// TwinCAT 3 PLC project PLC
// ProgramVersion: 3.1.4023.0
// libraries:
//   Tc2_ControllerToolbox, * (Beckhoff Automation GmbH)
//   Tc2_MC2, * (Beckhoff Automation GmbH)
//   Tc2_ModbusRTU, * (Beckhoff Automation GmbH)
//   Tc2_ModbusSrv, * (Beckhoff Automation GmbH)
//   Tc2_SerialCom, * (Beckhoff Automation GmbH)
//   Tc2_Standard, * (Beckhoff Automation GmbH)
//   Tc2_System, * (Beckhoff Automation GmbH)
//   Tc2_Utilities, * (Beckhoff Automation GmbH)
//   Tc3_Module, * (Beckhoff Automation GmbH)
//   VisuDialogs, * (System)
//   VisuSymbols,3.5.10.0,System
// project tree:
//   DUTs/ DUT_MB.TcDUT, DUT_MBReads.TcDUT
//   / Fast.TcTTO, GlobalTextList.TcGTLO, PlcTask.TcTTO, Visualization Manager.TcVMO (not stored)
//   GVLs/ GVL.TcGVL
//   POUs/ Background.TcPOU, BackgroundEL.TcPOU, FB_CCMT4Setup.TcPOU, FB_FanModbus.TcPOU, FB_FanWriteReg.TcPOU, FB_FormatTempRTD.TcPOU, FB_FormatTempTC.TcPOU, FB_LedOff.TcPOU, FB_ModBusTCPReadRegs.TcPOU, FB_ValveModbus.TcPOU, FB_MoveStepperRel.TcPOU, FB_MoveStepperLoop.TcPOU, FB_MoveStepperAbs.TcPOU, FB_mVtoTemp.TcPOU, FB_PLoop.TcPOU, FB_SanityCheck.TcPOU, FB_SerialCom.TcPOU, FB_StepperCtrl.TcPOU, FB_ModBusTCPWriteRegs.TcPOU, MAIN.TcPOU
//   VISUs/ Visu_MAIN.TcVIS

CONFIGURATION PLC
    RESOURCE PLC ON TwinCAT3
        TASK Fast(INTERVAL := T#1ms, PRIORITY := 4);
        TASK PlcTask(INTERVAL := T#10ms, PRIORITY := 10);
        PROGRAM Background WITH Fast : Background;
        PROGRAM MAIN WITH PlcTask : MAIN;
    END_RESOURCE
END_CONFIGURATION

// ---- DUTs/DUT_MB.TcDUT
TYPE DUT_MB :
STRUCT
	
	bExecute	:BOOL;	
	bBusy		:BOOL;
	bError		:BOOL;
	nErrId		:UDINT;
	
END_STRUCT
END_TYPE

// ---- DUTs/DUT_MBReads.TcDUT
TYPE DUT_MBReads EXTENDS DUT_MB :
STRUCT
	cbRead:UDINT;
	
END_STRUCT
END_TYPE

// ---- GVLs/GVL.TcGVL
VAR_GLOBAL
	RxBufferEL_RTD				: ComBuffer;		(* Receive data buffer; used with all receive function blocks *)
	TxBufferEL_RTD				: ComBuffer;		(* Transmit data buffer; used with all receive function blocks *)
	RxBufferEL_TC				: ComBuffer;		(* Receive data buffer; used with all receive function blocks *)
	TxBufferEL_TC				: ComBuffer;		(* Transmit data buffer; used with all receive function blocks *)
	RxBufferEL_Flow				: ComBuffer;
	TxBufferEL_Flow				: ComBuffer;
	RxBufferEL_MB				: ComBuffer;
	TxBufferEL_MB				: ComBuffer;
	f_mbMaster					: ModbusRtuMaster_KL6x22B;
	
	MAX_CSV_ROWS 				: UDINT := 100;
	MAX_CSV_COLUMNS 			: UDINT := 5;
	MAX_CSV_FIELD_LENGTH		: UDINT := 100;
(*	
// AXIS 1 CONTROL VARIABLES
	bEnable1				 	: BOOL := FALSE;	(* Axis enabled state *)
	bMove_Absolute1			 	: BOOL := FALSE;	(* Starts an absolute motion *)
	bJogFwd1				 	: BOOL := FALSE;	(* Starts rotating the axis at constant speed with CW direction *)
	bJogBack1				 	: BOOL := FALSE;	(* Starts rotating the axis at constant speed with CCCW direction *)
	bReset1					 	: BOOL := FALSE;	(* Resets the axis *)
	bHalt1					 	: BOOL := FALSE;	(* Stops the axis *)
	bStop1					 	: BOOL := FALSE;	(* Stops the axis *)
	bestop1					 	: BOOL := TRUE;		(* ESTOP button status *)
	bMove_Jog1				 	: BOOL := FALSE;	(* Starts actual motion *)
	bJogC1					 	: BOOL := FALSE;	(* Final Jog flag *)
	position1 					: UDINT;
	
// AXIS 2 CONTROL VARIABLES
	bEnable2				 	: BOOL := FALSE;	(* Axis enabled state *)
	bMove_Absolute2			 	: BOOL := FALSE;	(* Starts an absolute motion *)
	bJogFwd2				 	: BOOL := FALSE;	(* Starts rotating the axis at constant speed with CW direction *)
	bJogBack2				 	: BOOL := FALSE;	(* Starts rotating the axis at constant speed with CCCW direction *)
	bReset2					 	: BOOL := FALSE;	(* Resets the axis *)
	bHalt2					 	: BOOL := FALSE;	(* Stops the axis *)
	bStop2					 	: BOOL := FALSE;	(* Stops the axis *)
	bestop2					 	: BOOL := TRUE;		(* ESTOP button status *)
	bMove_Jog2				 	: BOOL := FALSE;	(* Starts actual motion *)
	bJogC2					 	: BOOL := FALSE;	(* Final Jog flag *)
	position2 					: UDINT;
*)	
// RELAY CONTROL VARIABLES
	bRelay1	AT %Q*			 	: BOOL := FALSE;
	bRelay2	AT %Q*				: BOOL := FALSE;
	
// 4...20mA ANALOG INPUT VARIABLES
	aiPress01 AT %I*			: INT;
	aiPress02 AT %I*			: INT;	
	aiPress03 AT %I*			: INT;	
	aiPress04 AT %I*			: INT;
	aiHBX01 AT %I*				: INT;
	
// RTD TEMPERATURE VARIABLES
	rtd01						: INT;
	rtd02						: INT;
	
// 0-10V ANALOG INPUT VARIABLES
	flow01 AT %I*				: INT;
	aiV02	AT %I*				: INT;
	
// PID VARIABLES
	TargetPos AT %Q*			: LREAL;
	
// 2Ch RTD VARIABLES
	RTD2Ch1	AT %I*				: INT;
	RTD2Ch2	AT %I*				: INT;
	RTD2Ch3	AT %I*				: INT;
	RTD2Ch4	AT %I*				: INT;
	RTD2Ch5	AT %I*				: INT;
	RTD2Ch6	AT %I*				: INT;
	RTD2Ch7	AT %I*				: INT;
	RTD2Ch8	AT %I*				: INT;
	
// 4Ch RTD VARIABLES
	RTD4Ch1	AT %I*				: INT;
	
END_VAR

// ---- POUs/Background.TcPOU
PROGRAM Background
VAR
END_VAR

(*
The SerialLineControl function block is supposed to be called in every PLC cycle.
It communicates with the serial line hardware device and transmits or receives data.
The SerialLineControl can be called in the standard task (e.g.for PcCOM port usage) 
or in a separate fast task (e.g.for terminal usage) as well.
A fast separate task will be necessary at high baud rates or with KL6001 terminals 
which have a small process image (3 or 5 data bytes only)
*)

(* background communication with the EL6002 and EL6021 terminal *)
BackgroundEL();

END_PROGRAM

// ---- POUs/BackgroundEL.TcPOU
PROGRAM BackgroundEL
VAR
	(* background communication with the EL6021 terminal *)
	fbEL6021Ctrl_RTD			: SerialLineControl;
	bEL6021CtrlError_RTD		: BOOL;
	eEL6021CtrlErrorID_RTD		: ComError_t;
	(* 	I/O variables for a EL6021 terminal*)
	stIn_EL6001_RTD AT %I*		: EL6inData22B;	(* linked to the EL6001 in the TwinCAT System Manager *)
	stOut_EL6001_RTD AT %Q*		: EL6outData22B;(* linked to the EL6001 in the TwinCAT System Manager *)
	
	(* background communication with the EL6021 terminal *)
	fbEL6021Ctrl_TC			: SerialLineControl;
	bEL6021CtrlError_TC		: BOOL;
	eEL6021CtrlErrorID_TC		: ComError_t;
	(* 	I/O variables for a EL6021 terminal*)
	stIn_EL6001_TC AT %I*		: EL6inData22B;	(* linked to the EL6001 in the TwinCAT System Manager *)
	stOut_EL6001_TC AT %Q*		: EL6outData22B;(* linked to the EL6001 in the TwinCAT System Manager *)
	
	(* background communication with the EL6002 terminal *)
	fbEL6002Ctrl_Flow			: SerialLineControl;
	bEL6002CtrlError_Flow		: BOOL;
	eEL6002CtrlErrorID_Flow		: ComError_t;
	(* 	I/O variables for a EL6002 terminal*)
	stIn_EL6002_Flow AT %I*		: EL6inData22B;	(* linked to the EL6001 in the TwinCAT System Manager *)
	stOut_EL6002_Flow AT %Q*		: EL6outData22B;(* linked to the EL6001 in the TwinCAT System Manager *)
	
		(* background communication with the EL6002 terminal *)
	fbEL6002Ctrl_MB			: SerialLineControl;
	bEL6002CtrlError_MB		: BOOL;
	eEL6002CtrlErrorID_MB		: ComError_t;
	(* 	I/O variables for a EL6002 terminal*)
	stIn_EL6002_MB AT %I*		: EL6inData22B;	(* linked to the EL6001 in the TwinCAT System Manager *)

END_VAR
VAR_INPUT
		stOut_EL6002_MB AT %Q*		: EL6outData22B;(* linked to the EL6001 in the TwinCAT System Manager *)
END_VAR

(*
The SerialLineControl function block is supposed to be called in every PLC cycle.
It communicates with the serial line hardware device and transmits or receives data.
The SerialLineControl can be called in the standard task (e.g.for PcCOM port usage) 
or in a separate fast task (e.g.for terminal usage) as well.
A fast separate task will be necessary at high baud rates or with KL6001 terminals 
which have a small process image (3 or 5 data bytes only)
*)

(* background communication with the EL6021 terminal *)
fbEL6021Ctrl_RTD(
	Mode := SERIALLINEMODE_EL6_22B,
	pComIn := ADR(stIn_EL6001_RTD), 
	pComOut:= ADR(stOut_EL6001_RTD), 
	SizeComIn := SIZEOF(stIn_EL6001_RTD), 
	Error => bEL6021CtrlError_RTD, 
	ErrorID => eEL6021CtrlErrorID_RTD,
	TxBuffer := GVL.TxBufferEL_RTD, 
	RxBuffer := GVL.RxBufferEL_RTD );
IF fbEL6021Ctrl_RTD.Error THEN
	bEL6021CtrlError_RTD := TRUE;
	eEL6021CtrlErrorID_RTD := fbEL6021Ctrl_RTD.ErrorID;
END_IF

(* background communication with the EL6021 terminal *)
fbEL6021Ctrl_TC(
	Mode := SERIALLINEMODE_EL6_22B,
	pComIn := ADR(stIn_EL6001_TC), 
	pComOut:= ADR(stOut_EL6001_TC), 
	SizeComIn := SIZEOF(stIn_EL6001_TC), 
	Error => bEL6021CtrlError_TC, 
	ErrorID => eEL6021CtrlErrorID_TC,
	TxBuffer := GVL.TxBufferEL_TC, 
	RxBuffer := GVL.RxBufferEL_TC );
IF fbEL6021Ctrl_TC.Error THEN
	bEL6021CtrlError_TC := TRUE;
	eEL6021CtrlErrorID_TC := fbEL6021Ctrl_RTD.ErrorID;
END_IF

(* background communication with the EL6021 terminal *)
fbEL6002Ctrl_Flow(
	Mode := SERIALLINEMODE_EL6_22B,
	pComIn := ADR(stIn_EL6002_Flow), 
	pComOut:= ADR(stOut_EL6002_Flow), 
	SizeComIn := SIZEOF(stIn_EL6002_Flow), 
	Error => bEL6002CtrlError_Flow, 
	ErrorID => eEL6002CtrlErrorID_Flow,
	TxBuffer := GVL.TxBufferEL_Flow, 
	RxBuffer := GVL.RxBufferEL_Flow );
IF fbEL6002Ctrl_Flow.Error THEN
	bEL6002CtrlError_Flow := TRUE;
	eEL6002CtrlErrorID_Flow := fbEL6002Ctrl_Flow.ErrorID;
END_IF

(* background communication with the EL6021 terminal *)
fbEL6002Ctrl_MB(
	Mode := SERIALLINEMODE_EL6_22B,
	pComIn := ADR(stIn_EL6002_MB), 
	pComOut:= ADR(stOut_EL6002_MB), 
	SizeComIn := SIZEOF(stIn_EL6002_MB), 
	Error => bEL6002CtrlError_MB, 
	ErrorID => eEL6002CtrlErrorID_MB,
	TxBuffer := GVL.TxBufferEL_MB, 
	RxBuffer := GVL.RxBufferEL_MB );
IF fbEL6002Ctrl_MB.Error THEN
	bEL6002CtrlError_MB := TRUE;
	eEL6002CtrlErrorID_MB := fbEL6002Ctrl_MB.ErrorID;
END_IF

END_PROGRAM

// ---- POUs/MAIN.TcPOU
PROGRAM MAIN
VAR
	fbEL6021RTD				: FB_SerialCom;
	fbEL6021TC				: FB_SerialCom;
	fbEL6002Flow			: FB_SerialCom;
	fbEL6021_MB				: FB_SerialCom;
	fbDoesItWork			: FB_SanityCheck;
	fbFormatRTD				: FB_FormatTempRTD;
	fbFormatTC				: FB_FormatTempTC;
	fbmVtoTemp				: FB_mVtoTemp;
	fbLedOff				: FB_LedOff;
	error					: ComError_t;
	fbPID					: FB_Ploop;
//	fbCloseValve1			: FB_CloseValve;
	fbMoveAxis1Rel			: FB_MoveStepperRel;
	fbMoveAxis1Abs			: FB_MoveStepperAbs;
	fbStepperLoop			: FB_MoveStepperLoop;
	
// Modbus Fan Control Variables
	Fan1 					: FB_FanModbus; // FB for controlling Ebm Pabst Fan over Modbus
	fbCCMT4mb				: FB_ValveModbus;
	fbSetupCCMTmb			: FB_CCMT4Setup;
	bFanEnable				: BOOL;
	mbReadAddr				: WORD := 16#D000;
	mbWriteAddr 			: WORD := 16#D000;
	mbReadData				: WORD;
	mbWriteData 			: WORD;
	smbRPM					: STRING;
	mbRPM					: WORD;
	tachometerData 			: REAL;
	speedNominal 			: REAL;
	
// Stepper Variables
	bJogFwd					: BOOL;
	bJogBack				: BOOL;
	bJogDone				: BOOL;
	bValve1Closed			: BOOL;

// Modbus Valve Variables
	percentOD				: STRING;
	cmdOD					: REAL;
	btnMbActivate 			: BOOL := FALSE;
	ccmtPos					: WORD;
	sCCMTPos				: STRING;
	bSetupComplete			: BOOL := 0;

// Misc. Variables	
	sVaporQual				: STRING;
	sTemp01					: STRING;
	sTemp02					: STRING;
	sPress01				: STRING;
	sPress02				: STRING;
	sPress03				: STRING;
	sPress04				: STRING;
	SurfaceRTD1 			: STRING;
	SurfaceRTD2 			: STRING;
	sStepperGoTo			: STRING;
	sStepperNumSteps		: STRING;
	RTDorTC					: BOOL;
	
	bTest					: BOOL := FALSE;
	TEST					: BOOL := FALSE;

///////////////////////////////////////////////////////////////////////
//Function16
	_MBWriteRegs	:FB_MBWriteRegs;
	MBWriteRegs		:DUT_MB;
	ar2				:ARRAY[0..99] OF INT;
	
	//Function3
	_MBReadRegs		:FB_ModBusTCPReadRegs;
	MBReadRegs		:DUT_MBReads;
	ar1				:ARRAY[0..99] OF INT;
	
	sIPAddr:STRING(15):='192.168.000.001';



END_VAR
VAR_INPUT
	fbAxis1					: FB_StepperCtrl;
	fbAxis2					: FB_StepperCtrl;
	msgOutRTD				: STRING;
	msgOutTC				: STRING;
	msgOutFlow				: STRING;
	TempRaw					: STRING;
	MoveTo					: UDINT;
	StepsToMove				: UDINT;
	bMoveRelative			: BOOL := FALSE;
	bMoveAbsolute			: BOOL := FALSE;
END_VAR
VAR_OUTPUT
	bDirection				: BOOL;
END_VAR

///////////////////////////////////////////
// CLOSE VALVES ON STARTUP
///////////////////////////////////////////
//WHILE bValve1Closed <> TRUE DO
//	fbCloseValve1(bDone => bValve1Closed); 
//END_WHILE

// CCMT 4 Modbus Setup Routine
IF bSetupComplete = 0 THEN
	fbSetupCCMTmb(bSetupComplete => bSetupComplete);
END_IF


///////////////////////////////////////////
// CALL RS-485 ROUTINE
///////////////////////////////////////////
Background();

///////////////////////////////////////////
// RTD AND TC TEMP READINGS
///////////////////////////////////////////

fbEL6021RTD(
	TxBuffer := TxBufferEL_RTD,
	RxBuffer := RxBufferEL_RTD,
	msgOUT => msgOutRTD,
	prefix := '°C',
	suffix := ','
);

fbFormatRTD(
	sTempRaw := msgOutRTD, 
);
	
fbEL6021TC(
	TxBuffer := TxBufferEL_TC,
	RxBuffer := RxBufferEL_TC,
	msgOUT => msgOutTC,
	prefix := 'mV',
	suffix := ','
);
	
fbFormatTC(
	sTempRaw := msgOutTC
);

fbmVtoTemp(mVtempArray := fbFormatTC.tempArray);
fbmVtoTemp(T_cj := (INT_TO_LREAL(GVL.RTD4Ch1) / 10));

///////////////////////////////////////////
// FLOW METER RS-232
///////////////////////////////////////////

fbEL6002Flow(
	TxBuffer := TxBufferEL_Flow,
	RxBuffer := RxBufferEL_Flow,
	msgOUT => msgOutFlow,
	prefix := ,//'$N',
	suffix := //'$R'
);

///////////////////////////////////////////
// CALL BLINKENLIGHTS SANITY CHECK
///////////////////////////////////////////
fbDoesItWork();

///////////////////////////////////////////
// CALL VALVE PID CONTROL
///////////////////////////////////////////
fbPID(
		fSetPointValue := 100
);

///////////////////////////////////////////
// FORMAT AHU BOARD DATA FOR GUI
///////////////////////////////////////////
sVaporQual := TO_STRING(20 - 16 * (INT_TO_REAL(GVL.aiHBX01) / 32767));
sPress01 := TO_STRING(100 * (INT_TO_REAL((GVL.aiPress01) * 2) / 65536));
sPress02 := TO_STRING(100 * (INT_TO_REAL((GVL.aiPress02) * 2) / 65536));
sPress03 := TO_STRING(100 * (INT_TO_REAL((GVL.aiPress03) * 2) / 65536));
sPress04 := TO_STRING(100 * (INT_TO_REAL((GVL.aiPress04) * 2) / 65536));
SurfaceRTD1 := TO_STRING(INT_TO_REAL(GVL.RTD2Ch1) / 10);
SurfaceRTD2 := TO_STRING(INT_TO_REAL(GVL.RTD2Ch2) / 10);

IF bJogFwd = TRUE THEN
	fbAxis1(bJogFwd := TRUE, bJogBack := FALSE, bJogDone => bJogDone);
END_IF

IF bJogBack = TRUE THEN
	fbAxis1(bJogBack := TRUE, bJogFwd := FALSE, bJogDone => bJogDone);
END_IF

IF (bJogFwd = FALSE AND bJogBack = FALSE) OR bJogDone = TRUE THEN
	fbAxis1(bJogFwd := FALSE, bJogBack := FALSE);
END_IF

IF bMoveRelative = TRUE THEN
	fbMoveAxis1Rel(
		stepsToMove := STRING_TO_INT(sStepperNumSteps)
	);
END_IF

IF bMoveAbsolute = TRUE THEN
	fbMoveAxis1Abs(
		stepsToMove := STRING_TO_INT(sStepperGoTo)
	);
END_IF

IF TEST = TRUE THEN
	fbStepperLoop(
		stepsToMove := STRING_TO_INT(sStepperGoTo)
	);
END_IF

///////////////////////////////////////////
// FAN CONTROL
///////////////////////////////////////////


IF bFanEnable = TRUE THEN
	Fan1(
	f_mbReadAddr := mbReadAddr,
	f_mbWriteAddr := mbWriteAddr,
	f_mbWriteData := mbWriteData,
	f_mbRPM := TO_WORD(smbRPM),
	//f_state := state,
	//f_nextState := nextState,
	f_mbReadData => mbReadData,
	f_tachometerData => tachometerData,
	f_speedNominal => speedNominal
);
ELSE
	Fan1(
	f_mbReadAddr := mbReadAddr,
	f_mbWriteAddr := mbWriteAddr,
	f_mbWriteData := mbWriteData,
	f_mbRPM := 0,
	//f_state := state,
	//f_nextState := nextState,
	f_mbReadData => mbReadData,
	f_tachometerData => tachometerData,
	f_speedNominal => speedNominal
);
END_IF

// CCMT 4 Modbus Control

cmdOD := ((STRING_TO_REAL(percentOD) / 1100) * 1000);
IF STRING_TO_REAL(percentOD) > 1100 THEN
	percentOD := '1100';
END_IF
IF cmdOD > 1000 THEN
	cmdOD := 1000;
END_IF
IF cmdOD < 0 THEN
	cmdOD := 0;
END_IF

IF btnMbActivate = TRUE THEN
	fbCCMT4mb(
		posData := REAL_TO_WORD(cmdOD),
		posActualData => ccmtPos
		);
		sCCMTPos := WORD_TO_STRING(ccmtPos);
ELSE
	fbCCMT4mb(
		posData := 0,
		posActualData => ccmtPos
		);
		sCCMTPos := WORD_TO_STRING(ccmtPos);
END_IF

fbLedOff();
fbEL6021_MB(
	RxBuffer := GVL.RxBufferEL_MB, 
	TxBuffer := GVL.TxBufferEL_MB
);

END_PROGRAM

// ---- POUs/FB_SerialCom.TcPOU
FUNCTION_BLOCK FB_SerialCom
VAR_IN_OUT
	TxBuffer			: ComBuffer;
	RxBuffer			: ComBuffer;
END_VAR
VAR
	fbReceive			: ReceiveString;

	sReceivedString		: STRING;
	sLastReceivedString	: STRING;
	bStringReceived		: BOOL;
	bReceiveBusy		: BOOL;
	bReceiveError		: BOOL;
	eReceiveErrorID		: ComError_t;
	bReceiveTimeout		: BOOL;
	pSendData : POINTER TO BYTE;
    Length : UDINT;
END_VAR
VAR_INPUT
	prefix				: STRING;
	suffix				: STRING;
	fbSendData			: SendData;
END_VAR
VAR_OUTPUT
	msgOUT				: STRING;
	errorID				: ComError_t;
	Busy 				: BOOL;
    Error 				: ComError_t;
END_VAR

//	Receive string data:
//	The block receives any data strings beginning with a STX ($02) and ending with an ETX ($03) character.	

fbReceive(
	Prefix := prefix,
	Suffix := suffix,
	Timeout := T#1S,
	ReceivedString := msgOUT,
	RXbuffer := RxBuffer,
	StringReceived => bStringReceived,
	Busy => bReceiveBusy,
	Error => errorID,
	RxTimeout => bReceiveTimeout );
IF fbReceive.Error <> COMERROR_NOERROR THEN
	eReceiveErrorID := fbReceive.Error;
END_IF

fbSendData(
	pSendData := ADR(pSendData),
	Length := SIZEOF(pSendData),
	Busy => Busy,
	Error => Error,
	TXBuffer := GVL.TxBufferEL_MB
	);

END_FUNCTION_BLOCK

// ---- POUs/FB_SanityCheck.TcPOU
FUNCTION_BLOCK FB_SanityCheck
VAR_INPUT
END_VAR
VAR_OUTPUT
END_VAR
VAR
	Delay 			: TON;
	step			: INT := 1;
	out1 AT %Q* 	: BOOL;
	out2 AT %Q*		: BOOL;
	out3 AT %Q*		: BOOL;
	out4 AT %Q*		: BOOL;
	out5 AT %Q*		: BOOL;
	out6 AT %Q*		: BOOL;
	out7 AT %Q*		: BOOL;
	out8 AT %Q*		: BOOL;
END_VAR

CASE step OF
1:
	IF out1 = FALSE THEN
		out1 := TRUE;
		ELSE
			out1 := FALSE; 
	END_IF
	
	Delay(IN:=TRUE, PT:=T#1S);
	IF NOT(Delay.Q) THEN
  		RETURN;
	END_IF
	
	Delay(IN:=FALSE);
	
	step := step + 1;

2:
	IF out2 = FALSE THEN
		out2 := TRUE;
		ELSE
			out2 := FALSE;
	END_IF
	
	Delay(IN:=TRUE, PT:=T#1S);
	
	IF NOT(Delay.Q) THEN
    	RETURN;
	END_IF
	
	Delay(IN:=FALSE);
	
	step := step + 1;
	
3:
	IF out3 = FALSE THEN
		out3 := TRUE;
		ELSE
			out3 := FALSE;
	END_IF
	
	Delay(IN:=TRUE, PT:=T#1S);
	
	IF NOT(Delay.Q) THEN
   		RETURN;
	END_IF
	
	Delay(IN:=FALSE);

	step := step + 1;
	
4:
	IF out4 = FALSE THEN
		out4 := TRUE;
		ELSE
			out4 := FALSE;
	END_IF
	
	Delay(IN:=TRUE, PT:=T#1S);
	
	IF NOT(Delay.Q) THEN
    	RETURN;
	END_IF
	
	Delay(IN:=FALSE);
	
	step := step + 1;
	
5:
	IF out5 = FALSE THEN
		out5 := TRUE;
		ELSE
			out5 := FALSE;
	END_IF
	
	Delay(IN:=TRUE, PT:=T#1S);
	
	IF NOT(Delay.Q) THEN
    	RETURN;
	END_IF
	
	Delay(IN:=FALSE);
	
	step := step + 1;
	
6:
	IF out6 = FALSE THEN
		out6 := TRUE;
		ELSE
			out6 := FALSE;
	END_IF
	
	Delay(IN:=TRUE, PT:=T#1S);
	
	IF NOT(Delay.Q) THEN
    	RETURN;
	END_IF

	Delay(IN:=FALSE);

	step := step + 1;
	
7:
	IF out7 = FALSE THEN
		out7 := TRUE;
		ELSE
			out7 := FALSE;
	END_IF
	
	Delay(IN:=TRUE, PT:=T#1S);
	
	IF NOT(Delay.Q) THEN
    	RETURN;
	END_IF

	Delay(IN:=FALSE);

	step := step + 1;
	
8:
	IF out8 = FALSE THEN
		out8 := TRUE;
		ELSE
			out8 := FALSE;
	END_IF
	
	Delay(IN:=TRUE, PT:=T#1S);
	
	IF NOT(Delay.Q) THEN
    	RETURN;
	END_IF
	
	Delay(IN:=FALSE);

	step := 1;
	
END_CASE

END_FUNCTION_BLOCK

// ---- POUs/FB_FormatTempRTD.TcPOU
FUNCTION_BLOCK FB_FormatTempRTD
VAR_INPUT
	sTempRaw 			: STRING;
END_VAR
VAR_OUTPUT
END_VAR
VAR
	RTDarray			: ARRAY[0..9] OF STRING;
	ArrayPos			: INT := 1;
END_VAR

(*
sArrayPos := MID(sTempRaw, 2, 3);
IF sArrayPos <> '' THEN
	ArrayPos := TO_INT(MID(sTempRaw, 2, 3)); // Find what temperature value is being read from string
	ArrayPos := ArrayPos - 1;

	RTDarray[ArrayPos] := MID(sTempRaw, 11, 6);
END_IF
*)
(*
// If string value is first value (presents w/ '$R$N'), extract both the 31st and 0th temperature value
IF FIND(sTempRaw, '$R$N') > 0 THEN
	tempArray[9] := MID(sTempRaw, 10, 6);
	tempArray[0] := RIGHT(sTempRaw, 11);
ELSE
	ArrayPos := STRING_TO_INT(MID(sTempRaw, 2, 3)); // Find what temperature value is being read from string
	
	IF INT_TO_STRING(ArrayPos) <> '00' THEN // If its the 0th, ignore to avoid duplicate read with spurious value
		tempArray[TO_INT(ArrayPos)] := MID(sTempRaw, 10, 6);
	END_IF
END_IF
*)

IF FIND(sTempRaw, '°C01') > 0 THEN
	ArrayPos := FIND(sTempRaw, '°C01');
	RTDarray[0] := MID(sTempRaw, 11, ArrayPos + 5);
END_IF
IF FIND(sTempRaw, '°C02') > 0 THEN
	ArrayPos := FIND(sTempRaw, '°C02');
	RTDarray[1] := MID(sTempRaw, 11, ArrayPos + 5);
END_IF
IF FIND(sTempRaw, '°C03') > 0 THEN
	ArrayPos := FIND(sTempRaw, '°C03');
	RTDarray[2] := MID(sTempRaw, 11, ArrayPos + 5);
END_IF
IF FIND(sTempRaw, '°C04') > 0 THEN
	ArrayPos := FIND(sTempRaw, '°C04');
	RTDarray[3] := MID(sTempRaw, 11, ArrayPos + 5);
END_IF
IF FIND(sTempRaw, '°C05') > 0 THEN
	ArrayPos := FIND(sTempRaw, '°C05');
	RTDarray[4] := MID(sTempRaw, 11, ArrayPos + 5);
END_IF
IF FIND(sTempRaw, '°C06') > 0 THEN
	ArrayPos := FIND(sTempRaw, '°C06');
	RTDarray[5] := MID(sTempRaw, 11, ArrayPos + 5);
END_IF
IF FIND(sTempRaw, '°C07') > 0 THEN
	ArrayPos := FIND(sTempRaw, '°C07');
	RTDarray[6] := MID(sTempRaw, 11, ArrayPos + 5);
END_IF
IF FIND(sTempRaw, '°C08') > 0 THEN
	ArrayPos := FIND(sTempRaw, '°C08');
	RTDarray[7] := MID(sTempRaw, 11, ArrayPos + 5);
END_IF
IF FIND(sTempRaw, '°C09') > 0 THEN
	ArrayPos := FIND(sTempRaw, '°C09');
	RTDarray[8] := MID(sTempRaw, 11, ArrayPos + 5);
END_IF
IF FIND(sTempRaw, '°C10') > 0 THEN
	ArrayPos := FIND(sTempRaw, '°C10');
	RTDarray[9] := MID(sTempRaw, 11, ArrayPos + 5);
END_IF

END_FUNCTION_BLOCK

// ---- POUs/FB_FormatTempTC.TcPOU
FUNCTION_BLOCK FB_FormatTempTC
VAR_INPUT
	sTempRaw 			: STRING;
END_VAR
VAR_OUTPUT
	tempArray 			: ARRAY[0..31] OF STRING;
END_VAR
VAR
	ArrayPos 			: STRING;
	subString			: STRING;
END_VAR

// If string value is first value (presents w/ '$R$N'), extract both the 31st and 0th temperature value
IF FIND(sTempRaw, '$R$N') > 0 THEN
	tempArray[31] := MID(sTempRaw, 10, 6);
	tempArray[0] := RIGHT(sTempRaw, 11);
ELSE
	ArrayPos := MID(sTempRaw, 2, 3); // Find what temperature value is being read from string
	
	IF ArrayPos <> '00' THEN // If its the 0th, ignore to avoid duplicate read with spurious value
		tempArray[TO_INT(ArrayPos)] := MID(sTempRaw, 10, 6);
	END_IF
END_IF

END_FUNCTION_BLOCK

// ---- POUs/FB_mVtoTemp.TcPOU
FUNCTION_BLOCK FB_mVtoTemp
VAR
	Index					: INT := 0;
	test					: STRING;
	
// Constants for t < 0
	t0_1					: LREAL := -6.0000000E+01;
	v0_1					: LREAL := -2.1528350E+00;
	p1_1					: LREAL := 3.0449332E+01;
	p2_1					: LREAL := -1.2946560E+00;
	p3_1					: LREAL := -3.0500735E+00;
	p4_1					: LREAL := -1.9226856E-01;
	q1_1					: LREAL := 6.9877863E-03;
	q2_1					: LREAL := -1.0596207E-01;
	q3_1					: LREAL := -1.0774995E-02;

// Constants for t >= 0
	t0_2					: LREAL := 1.3500000E+02;
	v0_2					: LREAL := 5.9588600E+00;
	p1_2					: LREAL := 2.0325591E+01;
	p2_2					: LREAL := 3.3013079E+00;
	p3_2					: LREAL := 1.2638462E-01;
	p4_2					: LREAL := -8.2883695E-04;
	q1_2					: LREAL := 1.7595577E-01;
	q2_2					: LREAL := 7.9740521E-03;
	q3_2					: LREAL := 0;
	
// Cold junction compensation constants	
	v_cj					: LREAL;
	
	t0_cj					: LREAL := 2.5000000E+01;
	v0_cj					: LREAL := 9.9198279E-01;
	p1_cj					: LREAL := 4.0716564E-02;
	p2_cj					: LREAL := 7.1170297E-04;
	p3_cj					: LREAL := 6.8782631E-07;
	p4_cj					: LREAL := 4.3295061E-11;
	q1_cj					: LREAL := 1.6458102E-02;
	q2_cj					: LREAL := 0.0000000E+00;
	
	Vtc						: LREAL;
	Vm						: LREAL;
END_VAR
VAR_INPUT
	mVtempArray 			: ARRAY[0..31] OF STRING;
	sResult					: STRING;
	T_cj					: LREAL;
END_VAR
VAR_OUTPUT
	degCtempArray			: ARRAY[0..31] OF STRING;
	degCtemp				: STRING;
END_VAR

Vm := STRING_TO_REAL(mVtempArray[Index]);
v_cj := (v0_cj + (T_cj - t0_cj) * (p1_cj + (T_cj - t0_cj) )* (p2_cj + (T_cj - t0_cj) * (p3_cj + p4_cj * (T_cj - t0_cj)))) / (1 + (T_cj - t0_cj) * (q1_cj + q2_cj * (T_cj - t0_cj))); 
Vtc := Vm;// + v_cj;
	
IF Vtc < 0 THEN		
	degCtempArray[Index] := LREAL_TO_FMTSTR(t0_1 + ((((Vtc - v0_1) *(p1_1 + (Vtc - v0_1) *(p2_1 + (Vtc - v0_1) * (p3_1 + p4_1 * (Vtc - v0_1)))))) / ((1 + (Vtc - v0_1) *(q1_1 + (Vtc - v0_1) *(q2_1 + q3_1 * (Vtc - v0_1)))))), 6 , TRUE);
ELSE
	degCtempArray[Index] := LREAL_TO_FMTSTR(t0_2 + ((((Vtc - v0_2) *(p1_2 + (Vtc - v0_2) *(p2_2 + (Vtc - v0_2) * (p3_2 + p4_2 * (Vtc - v0_2)))))) / ((1 + (Vtc - v0_2) *(q1_2 + (Vtc - v0_2) *(q2_2 + q3_2 * (Vtc - v0_2)))))), 6, TRUE);
END_IF

Index := Index + 1;
IF Index > 31 THEN
	Index := 0;
END_IF

(*
mV := STRING_TO_REAL(test);
IF mv < 0 THEN		
	degCtemp := LREAL_TO_FMTSTR(t0_1 + ((((mV - v0_1) *(p1_1 + (mV - v0_1) *(p2_1 + (mV - v0_1) *(p3_1 + p4_1 * (mV - v0_1)))))) / ((1 + (mV - v0_1) *(q1_1 + (mV - v0_1) *(q2_1 + q3_1 * (mV - v0_1)))))), 6 , TRUE);
ELSE
	degCtemp := LREAL_TO_FMTSTR(t0_2 + ((((mV - v0_2) *(p1_2 + (mV - v0_2) *(p2_2 + (mV - v0_2) *(p3_2 + p4_2 * (mV - v0_2)))))) / ((1 + (mV - v0_2) *(q1_2 + (mV - v0_2) *(q2_2 + q3_2 * (mV - v0_2)))))), 6, TRUE);
END_IF
*)

END_FUNCTION_BLOCK

// ---- POUs/FB_LedOff.TcPOU
FUNCTION_BLOCK FB_LedOff
VAR_INPUT
END_VAR
VAR_OUTPUT
END_VAR
VAR
	state : INT := 0;
	fbSerialSend : FB_SerialCom;
	d0 : BYTE := 16#01;
	d1 : BYTE := 16#44;
	d2 : BYTE := 16#00;
	d3 : BYTE := 16#13;
	d4 : BYTE := 16#00;
	fbSendData : SendData;
END_VAR

(*
BackGroundEL.stOut_EL6002_MB.D[0] := 16#01;
BackGroundEL.stOut_EL6002_MB.D[1] := 16#44;
BackGroundEL.stOut_EL6002_MB.D[2] := 16#00;
BackGroundEL.stOut_EL6002_MB.D[3] := 16#13;
BackGroundEL.stOut_EL6002_MB.D[4] := 16#00;
*)
(*
CASE state OF 
0:
fbSerialSend(
	TxBuffer := GVL.TxBufferEL_MB,
	RxBuffer := GVL.RxBufferEL_MB,
	fbSendData := fbSendData.pSendData,
	Busy =>,
	Error =>
	);
	IF fbSerialSend.Busy = FALSE THEN
		state := state + 1;
	END_IF
1:
fbSerialSend(
	TxBuffer := GVL.TxBufferEL_MB,
	RxBuffer := GVL.RxBufferEL_MB,
	fbSendData := d0,
	Busy =>,
	Error =>
	);
	IF fbSerialSend.Busy = FALSE THEN
		state := state + 1;
	END_IF
2:
fbSerialSend(
	TxBuffer := GVL.TxBufferEL_MB,
	RxBuffer := GVL.RxBufferEL_MB,
	fbSendData := d0,
	Busy =>,
	Error =>
	);
	IF fbSerialSend.Busy = FALSE THEN
		state := state + 1;
	END_IF
3:
fbSerialSend(
	TxBuffer := GVL.TxBufferEL_MB,
	RxBuffer := GVL.RxBufferEL_MB,
	fbSendData := d0,
	Busy =>,
	Error =>
	);
	IF fbSerialSend.Busy = FALSE THEN
		state := state + 1;
	END_IF
4:
fbSerialSend(
	TxBuffer := GVL.TxBufferEL_MB,
	RxBuffer := GVL.RxBufferEL_MB,
	fbSendData := d0,
	Busy =>,
	Error =>
	);
	IF fbSerialSend.Busy = FALSE THEN
		state := 0;
	END_IF
END_CASE
*)

END_FUNCTION_BLOCK

// ---- POUs/FB_PLoop.TcPOU
FUNCTION_BLOCK FB_PLoop
VAR_INPUT
	fSetpointValue					: REAL ;
END_VAR
VAR_OUTPUT
END_VAR
VAR
	fbPID : FB_CTRL_PID;
	stCTRL_PID_PARAMS				: ST_CTRL_PID_PARAMS;
	eErrorId						: E_CTRL_ERRORCODES;
	eMode							: E_CTRL_MODE;
	//fActualValue					: REAL;
	fManSyncValue					: REAL;
	fOut							: LREAL;
	//pos_offset						: REAL ;
	//pos_cmd							: REAL ;
	//mir_adjusted					: REAL;
	bHold							: BOOL;
	bError							: BOOL;
	bARWactive						: BOOL;
	bSync							: BOOL;
	bInit							: BOOL	:= TRUE;
END_VAR

IF bInit THEN
	(* init parameter struct *)
	stCTRL_PID_PARAMS.tCtrlCycleTime		:= T#10ms;
	stCTRL_PID_PARAMS.tTaskCycleTime		:= T#10ms;
	stCTRL_PID_PARAMS.fKp					:= 5000.0;			(* proportional gain Kp				*)
	stCTRL_PID_PARAMS.tTn					:= T#0MS;			(*  Tn								*)
	stCTRL_PID_PARAMS.tTv					:= T#0MS;			(*  Tv								*)
	stCTRL_PID_PARAMS.tTd					:= T#0S;			(*  Td								*)
	stCTRL_PID_PARAMS.fOutMaxLimit			:= (10921800);	(* maximum output limit				*)
	stCTRL_PID_PARAMS.fOutMinLimit			:= (-10921800);	(* minimum output limit				*)
	stCTRL_PID_PARAMS.bDInTheFeedbackPath	:= FALSE;
	stCTRL_PID_PARAMS.bDInTheFeedbackPath	:= FALSE;
	stCTRL_PID_PARAMS.bARWOnIPartOnly		:= TRUE;

	(* set the mode to ACTIVE --> normal operation *)
	eMode := eCTRL_MODE_ACTIVE;

	(* reset the init flag *)
	bInit := FALSE;
END_IF

(* call controller *)
fbPID(			fSetpointValue		:= fSetpointValue ,
				fActualValue		:= GVL.aiHBX01,
				fManSyncValue		:= fManSyncValue,
				bSync				:= bSync,
				eMode				:= eMode,
				bHold				:= bHold,
				stParams			:= stCTRL_PID_PARAMS,
				fOut				=> fOut,
				bARWactive			=> bARWactive,
				eErrorId			=> eErrorId,
				bError				=> bError
				);
				
//GVL.target_vel := TO_DINT(fbPID.fOut);

END_FUNCTION_BLOCK

// ---- POUs/FB_MoveStepperRel.TcPOU
FUNCTION_BLOCK FB_MoveStepperRel
VAR_INPUT
	stepsToMove				: INT;
	PosCurrent				: UDINT;
END_VAR
VAR_OUTPUT
END_VAR
VAR
	Step 					: INT := 0;
	bPowerOn				: INT;
END_VAR

MAIN.fbAxis1.bEnable := TRUE;

CASE Step OF
0:
	//MAIN.fbAxis1.moveRelDist := 0.0;
	//MAIN.fbAxis1.moveRelVel := 0.0;
	//MAIN.fbAxis1.bMoveRelExe := FALSE;
	MAIN.fbAxis1.bHaltExe := FALSE;
	Step := 1;
1:

	IF MAIN.fbAxis1.bPwrStatus THEN
		MAIN.fbAxis1.moveRelDist := stepsToMove;
		MAIN.fbAxis1.moveRelVel := 100;
		MAIN.fbAxis1.bMoveRelExe := TRUE;
		IF MAIN.fbAxis1.bMoveRelDone THEN
			MAIN.fbAxis1.bMoveRelExe := FALSE;
			MAIN.fbAxis1.bHaltExe := TRUE;
			Step := 2;
		END_IF
	END_IF	
2:
	IF MAIN.fbAxis1.bHaltDone = TRUE THEN
		MAIN.fbAxis1.bHaltExe := FALSE;
	END_IF

	MAIN.bMoveRelative := FALSE;
	
	Step := 0;
END_CASE

END_FUNCTION_BLOCK

// ---- POUs/FB_MoveStepperAbs.TcPOU
FUNCTION_BLOCK FB_MoveStepperAbs
VAR_INPUT
	stepsToMove				: INT;
	PosCurrent				: UDINT;
END_VAR
VAR_OUTPUT
END_VAR
VAR
	Step 					: INT := 0;
	bPowerOn				: INT;

END_VAR

MAIN.fbAxis1.bEnable := TRUE;

CASE Step OF
0:
	MAIN.fbAxis1.moveAbsPosition := 0.0;
	MAIN.fbAxis1.moveAbsVel := 0.0;
	MAIN.fbAxis1.bMoveAbsExe := FALSE;
	MAIN.fbAxis1.bHaltExe := FALSE;
	Step := 1;
1:

	IF MAIN.fbAxis1.bPwrStatus THEN
		MAIN.fbAxis1.moveAbsPosition := stepsToMove;
		MAIN.fbAxis1.moveAbsVel := 100;
		MAIN.fbAxis1.bMoveAbsExe := TRUE;
		IF MAIN.fbAxis1.bMoveAbsDone THEN
			MAIN.fbAxis1.bMoveAbsExe := FALSE;
			MAIN.fbAxis1.bHaltExe := TRUE;
			Step := 2;
		END_IF
	END_IF	
2:
	IF MAIN.fbAxis1.bHaltDone = TRUE THEN
		MAIN.fbAxis1.bHaltExe := FALSE;
	END_IF

	MAIN.bMoveAbsolute := FALSE;
	
	Step := 0;
END_CASE

END_FUNCTION_BLOCK

// ---- POUs/FB_MoveStepperLoop.TcPOU
FUNCTION_BLOCK FB_MoveStepperLoop
VAR_INPUT
	stepsToMove				: INT;
	PosCurrent				: UDINT;
END_VAR
VAR_OUTPUT
END_VAR
VAR
	Step 					: INT := 0;
	bPowerOn				: INT;
END_VAR

MAIN.fbAxis1.bEnable := TRUE;

CASE Step OF
0:
	MAIN.fbAxis1.moveRelDist := 0.0;
	MAIN.fbAxis1.moveRelVel := 0.0;
	MAIN.fbAxis1.bMoveRelExe := FALSE;
	MAIN.fbAxis1.bHaltExe := FALSE;
	Step := 1;
1:

	IF MAIN.fbAxis1.bPwrStatus THEN
		MAIN.fbAxis1.moveRelDist := 1;
		MAIN.fbAxis1.moveRelVel := 100;
		MAIN.fbAxis1.bMoveRelExe := TRUE;
		IF MAIN.fbAxis1.bMoveRelDone THEN
			MAIN.fbAxis1.bMoveRelExe := FALSE;
			MAIN.fbAxis1.bHaltExe := TRUE;
		END_IF
	END_IF
	StepsToMove := StepsToMove - 1;
	Step := 2;
2:
	IF MAIN.fbAxis1.bHaltDone = TRUE THEN
		MAIN.fbAxis1.bHaltExe := FALSE;
	END_IF

	MAIN.bMoveRelative := FALSE;
	IF StepsToMove = 0 THEN
		Step := 3;
	ELSE
		Step := 0;
	END_IF
END_CASE

END_FUNCTION_BLOCK

// ---- POUs/FB_FanModbus.TcPOU
FUNCTION_BLOCK FB_FanModbus
VAR_INPUT
	f_state						: UINT ;//:= 0;
	f_nextState					: UINT ;//:= 0;
	f_mbReadAddr				: WORD ;//:= 16#D000;
	f_mbWriteAddr 				: WORD ;//:= 16#D000;
	f_mbWriteData 				: WORD;
	f_mbRPM						: WORD;
END_VAR
VAR_OUTPUT
	f_tachometerData 			: REAL;
	f_mbReadData				: WORD;
	f_speedNominal 				: WORD;	
END_VAR
VAR
	f_mbMaster					: ModbusRtuMaster_KL6x22B;
	idx							: WORD;
	f_mbInputAddr 				: WORD;//:= 16#D000;
	f_mbInputData 				: WORD;
	f_mbUnit					: BYTE := 1;
	f_mbErrorId					: MODBUS_ERRORS;
	f_mbErrorFlag				: BOOL;
	f_mbBusy					: BOOL;
	f_mbBytesRec				: UINT;
	f_inputs					: ARRAY [0..1, 16#00 .. 16#26] OF UINT;
END_VAR

CASE f_state OF
0: // init, reset
	FOR idx := 0 TO 16#26 DO
		f_inputs[0, idx] := 16#D000 + idx;
	END_FOR
	f_mbInputAddr := 16#D010;
	idx := 0;
	f_nextState := 1;
	f_state := 1;

1: // read input registers
	f_mbMaster.ReadInputRegs(
		UnitID:= f_mbUnit, 
		Quantity:= 1, 
		MBAddr:= 16#D010,//f_mbInputAddr, 
		cbLength:= SIZEOF(f_mbInputData), 
		pMemoryAddr:= ADR(f_mbInputData), 
		Execute:= TRUE, 
		Timeout:= T#1S, 
		BUSY=> f_mbBusy, 
		Error=> f_mbErrorFlag, 
		ErrorId=> f_mbErrorId, 
		cbRead=> f_mbBytesRec
	);

	// if not busy, move to next input register
	IF f_mbBusy = FALSE THEN
		f_inputs[1, 16#10] := f_mbInputData;
		f_mbInputAddr := 16#D010;//f_mbInputAddr + 1;
		//idx := idx + 1;
		//IF idx > 16#26 THEN
		//	idx := 0;
		//	f_mbInputAddr := 16#D000;
		//END_IF
		
		//Read tachometer data. This is not the fastest 
		//sampling rate of the actual speed value, since
		//it is only measured once every 26 cycles.
		f_tachometerData := (f_inputs[1,16#10] * 16#802) / 16#FA00;
		
		// reset comms and go to next state
		f_mbMaster.ReadInputRegs(Execute := FALSE);
		f_state := f_nextState;
		// catch error
		IF f_mbErrorFlag = TRUE THEN
			f_state := 4;
		END_IF
	END_IF
	
2: // read holding register
	f_mbMaster.ReadRegs(
		UnitID:= f_mbUnit, 
		Quantity:= 1, 
		MBAddr:= f_mbReadAddr, 
		cbLength:= SIZEOF(f_mbReadData), 
		pMemoryAddr:= ADR(f_mbReadData), 
		Execute:= TRUE, 
		Timeout:= T#1S, 
		BUSY=> f_mbBusy, 
		Error=> f_mbErrorFlag, 
		ErrorId=> f_mbErrorId, 
		cbRead=> f_mbBytesRec
	);

	// read complete
	IF f_mbBusy = FALSE THEN
		// reset comms
		f_mbMaster.ReadRegs(Execute := FALSE);
		f_nextState := 1;
		f_state := f_nextState;
		// catch error
		IF f_mbErrorFlag = TRUE THEN
			f_state := 4;
		END_IF
	END_IF
	
3: // write register
	f_mbMaster.WriteSingleRegister(
		UnitID:= f_mbUnit, 
		Quantity:= 1, 
		MBAddr:= f_mbWriteAddr, 
		cbLength:= SIZEOF(f_mbWriteData), 
		pMemoryAddr:= ADR(f_mbWriteData), 
		Execute:= TRUE, 
		Timeout:= T#1S, 
		BUSY=> f_mbBusy, 
		Error=> f_mbErrorFlag, 
		ErrorId=> f_mbErrorId, 
		cbRead=> f_mbBytesRec
	);

	// write complete
	IF f_mbBusy = FALSE THEN
		// reset comms
		f_mbMaster.ReadRegs(Execute := FALSE);
		f_nextState := 1;
		f_state := f_nextState;
		// catch error
		IF f_mbErrorFlag = TRUE THEN
			f_state := 4;
		END_IF
	END_IF

4: // error, wait for reset

5: //RPM set
	f_mbWriteAddr := 16#D001 ;
	f_mbWriteData := ( f_mbRPM * 16#FA00 ) / 16#802;
	
	// write register
	f_mbMaster.WriteSingleRegister(
		UnitID:= f_mbUnit, 
		Quantity:= 1, 
		MBAddr:= f_mbWriteAddr, 
		cbLength:= SIZEOF(f_mbWriteData), 
		pMemoryAddr:= ADR(f_mbWriteData), 
		Execute:= TRUE, 
		Timeout:= T#1S, 
		BUSY=> f_mbBusy, 
		Error=> f_mbErrorFlag, 
		ErrorId=> f_mbErrorId, 
		cbRead=> f_mbBytesRec
	);

	// write complete
	IF f_mbBusy = FALSE THEN
		// reset comms
		f_mbMaster.ReadRegs(Execute := FALSE);
		f_nextState := 1;
		f_state := f_nextState;
		
		//Set RPM nominal output
		f_speedNominal := f_mbRPM;
		// catch error
		IF f_mbErrorFlag = TRUE THEN
			f_state := 4;
		END_IF
	END_IF

//NOTE need to add 
	
6:
	f_mbWriteAddr := 16#D001 ;
	f_mbWriteData := 16#0000 ;
	
	// write register
	f_mbMaster.WriteSingleRegister(
		UnitID:= f_mbUnit, 
		Quantity:= 1, 
		MBAddr:= f_mbWriteAddr, 
		cbLength:= SIZEOF(f_mbWriteData), 
		pMemoryAddr:= ADR(f_mbWriteData), 
		Execute:= TRUE, 
		Timeout:= T#1S, 
		BUSY=> f_mbBusy, 
		Error=> f_mbErrorFlag, 
		ErrorId=> f_mbErrorId, 
		cbRead=> f_mbBytesRec
	);

	// write complete
	IF f_mbBusy = FALSE THEN
		// reset comms
		f_mbMaster.ReadRegs(Execute := FALSE);
		f_nextState := 1;
		f_state := f_nextState;
		
		//Set RPM nominal output
		f_speedNominal := f_mbWriteData;
		// catch error
		IF f_mbErrorFlag = TRUE THEN
			f_state := 4;
		END_IF
	END_IF

ELSE // stop
	
END_CASE

END_FUNCTION_BLOCK

// ---- POUs/FB_ValveModbus.TcPOU
FUNCTION_BLOCK FB_ValveModbus
VAR_INPUT
	manMode						: WORD := 4035;
	manModeData					: WORD := 1;
	posMode						: WORD := 4036;
	posData						: WORD;
	posActual					: WORD:= 4067;
	f_state						: UINT := 1;
	f_nextState					: UINT;//:= 0;
	f_mbReadAddr				: WORD; //:= 4067;
	f_mbWriteAddr 				: WORD;//:= 16#D000;
	f_mbWriteData 				: WORD;
END_VAR
VAR_OUTPUT
	f_mbReadData				: WORD;
	posActualData				: WORD;
END_VAR
VAR
//	f_mbMaster					: ModbusRtuMaster_KL6x22B;
	idx							: WORD;
	f_mbInputAddr 				: WORD;//:= 16#D000;
	f_mbInputData 				: WORD;
	f_mbUnit					: BYTE := 1;
	f_mbErrorId					: MODBUS_ERRORS;
	f_mbErrorFlag				: BOOL;
	f_mbBusy					: BOOL;
	f_mbBytesRec				: UINT;
	f_inputs					: ARRAY [0..1, 16#00 .. 16#26] OF UINT;
END_VAR

CASE f_state OF

1: // write register
	GVL.f_mbMaster.WriteSingleRegister(
		UnitID:= f_mbUnit, 
		Quantity:= 1, 
		MBAddr:= manMode,//f_mbWriteAddr, 
		cbLength:= SIZEOF(manModeData), 
		pMemoryAddr:= ADR(manModeData), 
		Execute:= TRUE, 
		Timeout:= T#1S, 
		BUSY=> f_mbBusy, 
		Error=> f_mbErrorFlag, 
		ErrorId=> f_mbErrorId, 
		cbRead=> f_mbBytesRec
	);

	// write complete
	IF f_mbBusy = FALSE THEN
		// reset comms
		GVL.f_mbMaster.ReadRegs(Execute := FALSE);
		f_nextState := 3;
		f_state := f_nextState;
		// catch error
		IF f_mbErrorFlag = TRUE THEN
			f_state := 10;
		END_IF
	END_IF
2:
	f_nextState := 3;
	f_state := f_nextState;
3:
GVL.f_mbMaster.WriteSingleRegister(
		UnitID:= f_mbUnit, 
		Quantity:= 1, 
		MBAddr:= posMode, 
		cbLength:= SIZEOF(posData), 
		pMemoryAddr:= ADR(posData), 
		Execute:= TRUE, 
		Timeout:= T#1S, 
		BUSY=> f_mbBusy, 
		Error=> f_mbErrorFlag, 
		ErrorId=> f_mbErrorId, 
		cbRead=> f_mbBytesRec
	);

	// write complete
	IF f_mbBusy = FALSE THEN
		// reset comms
		GVL.f_mbMaster.ReadRegs(Execute := FALSE);
		f_nextState := 5;
		f_state := f_nextState;
		// catch error
		IF f_mbErrorFlag = TRUE THEN
			f_state := 10;
		END_IF
	END_IF
4:
	f_nextState := 5;
	f_state := f_nextState;
5:
GVL.f_mbMaster.ReadRegs(
		UnitID:= f_mbUnit, 
		Quantity:= 1, 
		MBAddr:= posActual, 
		cbLength:= SIZEOF(posActualData), 
		pMemoryAddr:= ADR(posActualData), 
		Execute:= TRUE, 
		Timeout:= T#1S, 
		BUSY=> f_mbBusy, 
		Error=> f_mbErrorFlag, 
		ErrorId=> f_mbErrorId, 
		cbRead=> f_mbBytesRec
	);

	// read complete
	IF f_mbBusy = FALSE THEN
		// reset comms
		GVL.f_mbMaster.ReadRegs(Execute := FALSE);
		f_nextState := 1;
		f_state := f_nextState;
		// catch error
		IF f_mbErrorFlag = TRUE THEN
			f_state := 10;
		END_IF
	END_IF
6:
	f_nextState := 1;
	f_state := f_nextState;
10:
	f_mbErrorFlag := FALSE;
	f_state := 1;

END_CASE

END_FUNCTION_BLOCK

// ---- POUs/FB_CCMT4Setup.TcPOU
FUNCTION_BLOCK FB_CCMT4Setup
VAR_INPUT
	mainSwitch					: WORD := 3000;
	mainSwitchData				: WORD;
	opMode						: WORD := 3001;
	opModeData					: WORD := 1;
	valveConfig					: WORD := 3131;
	valveConfigData				: WORD := 22;
	refrigerantType				: WORD := 3071;
	refrigerantTypeData			: WORD := 28;
	mbMainSwitch				: WORD := 4045;
	mbMainSwitchData			: WORD := 1;
	manMode						: WORD := 4035;
	manModeData					: WORD := 1;
	manModeTimeout				: WORD := 3176;
	manModeTimeoutData			: WORD := 3600;
	
	f_state						: UINT := 1;
	f_nextState					: UINT;//:= 0;
	f_mbReadAddr				: WORD; //:= 4067;
	f_mbWriteAddr 				: WORD;//:= 16#D000;
	f_mbWriteData 				: WORD;
END_VAR
VAR_OUTPUT
	f_mbReadData				: WORD;
	bSetupComplete				: BOOL := 0;
END_VAR
VAR
//	f_mbMaster					: ModbusRtuMaster_KL6x22B;
	idx							: WORD;
	f_mbInputAddr 				: WORD;//:= 16#D000;
	f_mbInputData 				: WORD;
	f_mbUnit					: BYTE := 1;
	f_mbErrorId					: MODBUS_ERRORS;
	f_mbErrorFlag				: BOOL;
	f_mbBusy					: BOOL;
	f_mbBytesRec				: UINT;
	f_inputs					: ARRAY [0..1, 16#00 .. 16#26] OF UINT;
END_VAR

CASE f_state OF

1: // write register
	mainSwitchData := 0;
	GVL.f_mbMaster.WriteSingleRegister(
		UnitID:= f_mbUnit, 
		Quantity:= 1, 
		MBAddr:= mainSwitch, 
		cbLength:= SIZEOF(mainSwitchData), 
		pMemoryAddr:= ADR(mainSwitchData), 
		Execute:= TRUE, 
		Timeout:= T#1S, 
		BUSY=> f_mbBusy, 
		Error=> f_mbErrorFlag, 
		ErrorId=> f_mbErrorId, 
		cbRead=> f_mbBytesRec
	);

	// write complete
	IF f_mbBusy = FALSE THEN
		// reset comms
		GVL.f_mbMaster.ReadRegs(Execute := FALSE);
		f_nextState := 2;
		f_state := f_nextState;
		// catch error
		IF f_mbErrorFlag = TRUE THEN
			f_state := 10;
		END_IF
	END_IF
2:
GVL.f_mbMaster.WriteSingleRegister(
		UnitID:= f_mbUnit, 
		Quantity:= 1, 
		MBAddr:= opMode, 
		cbLength:= SIZEOF(opModeData), 
		pMemoryAddr:= ADR(opModeData), 
		Execute:= TRUE, 
		Timeout:= T#1S, 
		BUSY=> f_mbBusy, 
		Error=> f_mbErrorFlag, 
		ErrorId=> f_mbErrorId, 
		cbRead=> f_mbBytesRec
	);

	// write complete
	IF f_mbBusy = FALSE THEN
		// reset comms
		GVL.f_mbMaster.ReadRegs(Execute := FALSE);
		f_nextState := 3;
		f_state := f_nextState;
		// catch error
		IF f_mbErrorFlag = TRUE THEN
			f_state := 10;
		END_IF
	END_IF
3:
GVL.f_mbMaster.ReadRegs(
		UnitID:= f_mbUnit, 
		Quantity:= 1, 
		MBAddr:= valveConfig, 
		cbLength:= SIZEOF(valveConfigData), 
		pMemoryAddr:= ADR(valveConfigData), 
		Execute:= TRUE, 
		Timeout:= T#1S, 
		BUSY=> f_mbBusy, 
		Error=> f_mbErrorFlag, 
		ErrorId=> f_mbErrorId, 
		cbRead=> f_mbBytesRec
	);

	// read complete
	IF f_mbBusy = FALSE THEN
		// reset comms
		GVL.f_mbMaster.ReadRegs(Execute := FALSE);
		f_nextState := 4;
		f_state := f_nextState;
		// catch error
		IF f_mbErrorFlag = TRUE THEN
			f_state := 10;
		END_IF
	END_IF
4:
	GVL.f_mbMaster.ReadRegs(
		UnitID:= f_mbUnit, 
		Quantity:= 1, 
		MBAddr:= refrigerantType, 
		cbLength:= SIZEOF(refrigerantTypeData), 
		pMemoryAddr:= ADR(refrigerantTypeData), 
		Execute:= TRUE, 
		Timeout:= T#1S, 
		BUSY=> f_mbBusy, 
		Error=> f_mbErrorFlag, 
		ErrorId=> f_mbErrorId, 
		cbRead=> f_mbBytesRec
	);

	// read complete
	IF f_mbBusy = FALSE THEN
		// reset comms
		GVL.f_mbMaster.ReadRegs(Execute := FALSE);
		f_nextState := 5;
		f_state := f_nextState;
		// catch error
		IF f_mbErrorFlag = TRUE THEN
			f_state := 10;
		END_IF
	END_IF
5:
	GVL.f_mbMaster.ReadRegs(
		UnitID:= f_mbUnit, 
		Quantity:= 1, 
		MBAddr:= mbMainSwitch, 
		cbLength:= SIZEOF(mbMainSwitchData), 
		pMemoryAddr:= ADR(mbMainSwitchData), 
		Execute:= TRUE, 
		Timeout:= T#1S, 
		BUSY=> f_mbBusy, 
		Error=> f_mbErrorFlag, 
		ErrorId=> f_mbErrorId, 
		cbRead=> f_mbBytesRec
	);

	// read complete
	IF f_mbBusy = FALSE THEN
		// reset comms
		GVL.f_mbMaster.ReadRegs(Execute := FALSE);
		f_nextState := 6;
		f_state := f_nextState;
		// catch error
		IF f_mbErrorFlag = TRUE THEN
			f_state := 10;
		END_IF
	END_IF
6:
GVL.f_mbMaster.ReadRegs(
		UnitID:= f_mbUnit, 
		Quantity:= 1, 
		MBAddr:= manMode, 
		cbLength:= SIZEOF(manModeData), 
		pMemoryAddr:= ADR(manModeData), 
		Execute:= TRUE, 
		Timeout:= T#1S, 
		BUSY=> f_mbBusy, 
		Error=> f_mbErrorFlag, 
		ErrorId=> f_mbErrorId, 
		cbRead=> f_mbBytesRec
	);

	// read complete
	IF f_mbBusy = FALSE THEN
		// reset comms
		GVL.f_mbMaster.ReadRegs(Execute := FALSE);
		f_nextState := 7;
		f_state := f_nextState;
		// catch error
		IF f_mbErrorFlag = TRUE THEN
			f_state := 10;
		END_IF
	END_IF
7:
GVL.f_mbMaster.ReadRegs(
		UnitID:= f_mbUnit, 
		Quantity:= 1, 
		MBAddr:= manModeTimeout, 
		cbLength:= SIZEOF(manModeTimeoutData), 
		pMemoryAddr:= ADR(manModeTimeoutData), 
		Execute:= TRUE, 
		Timeout:= T#1S, 
		BUSY=> f_mbBusy, 
		Error=> f_mbErrorFlag, 
		ErrorId=> f_mbErrorId, 
		cbRead=> f_mbBytesRec
	);

	// read complete
	IF f_mbBusy = FALSE THEN
		// reset comms
		GVL.f_mbMaster.ReadRegs(Execute := FALSE);
		f_nextState := 8;
		f_state := f_nextState;
		// catch error
		IF f_mbErrorFlag = TRUE THEN
			f_state := 10;
		END_IF
	END_IF
8:
	mainSwitchData := 1;
	GVL.f_mbMaster.ReadRegs(
		UnitID:= f_mbUnit, 
		Quantity:= 9, 
		MBAddr:= mainSwitch, 
		cbLength:= SIZEOF(mainSwitchData), 
		pMemoryAddr:= ADR(mainSwitchData), 
		Execute:= TRUE, 
		Timeout:= T#1S, 
		BUSY=> f_mbBusy, 
		Error=> f_mbErrorFlag, 
		ErrorId=> f_mbErrorId, 
		cbRead=> f_mbBytesRec
	);

	// read complete
	IF f_mbBusy = FALSE THEN
		// reset comms
		GVL.f_mbMaster.ReadRegs(Execute := FALSE);
		f_nextState := 9;
		f_state := f_nextState;
		// catch error
		IF f_mbErrorFlag = TRUE THEN
			f_state := 10;
		END_IF
	END_IF
9:
	bSetupComplete := 1;
10:

END_CASE

END_FUNCTION_BLOCK

// ---- POUs/FB_ModBusTCPReadRegs.TcPOU
FUNCTION_BLOCK FB_ModBusTCPReadRegs
VAR_INPUT
    sIPAddr    			: STRING(15);
    nTCPPort   			: UINT:= MODBUS_TCP_PORT;
    nUnitID    			: BYTE:=16#FF;
    nQuantity  			: WORD;
    nMBAddr    			: WORD;
    cbLength   			: UDINT;
    pDestAddr  			: POINTER TO BYTE;
    bExecute   			: BOOL;
    tTimeout   			: TIME;
END_VAR 
VAR_OUTPUT
    bBUSY      			: BOOL;
    bError     			: BOOL;
    nErrId     			: UDINT;
    cbRead     			: UDINT;
END_VAR 
VAR
    fbReadRegs        	: FB_MBReadRegs;
    bReadRegs         	: BOOL;
    bReadRegsBusy     	: BOOL;
    bReadRegsError    	: BOOL;
    nReadRegsErrorId  	: UDINT;
    nReadRegsCount    	: UDINT;
    arrData           	: ARRAY [1..2] OF WORD;
END_VAR

//Read the Regs from Modbus Server Function 3
fbReadRegs(
	sIPAddr := sIPAddr,					//Is a string containing the IP address of the target device
	nTCPPort := MODBUS_TCP_PORT,		//Port number of the target device
	nUnitID := 255,						//Identification number of a serial sub-network device, 16$FF if TCP/IP is used
	nQuantity := 10,					//Number of output registers (data words) to be read. The value of nQuantity must be > 0 
	nMBAddr := 0,						//Start address of the output registers to be read (word offset)
	cbLength := SIZEOF(arrData),		//Contains the max. byte size of the destination buffer. 
	pDestAddr := ADR(arrData),			//Contains the address of the destination buffer into which the data are to be read
	bExecute := fbReadRegs.bExecute,	//The function block is activated by a rising edge at this input
	tTimeout := T#1S,					//States the length of the timeout that may not be exceeded by execution of the ADS command
	bBusy => bBusy,							//When the function block is activated this output is set
	bError => bError,							//True if If an ADS error should occur during the transfer of the command
	nErrId => nErrId,							//Supplies the ADS error number when the bError output is set.
	cbRead => cbRead						//Contains the number of bytes currently read.
	);

END_FUNCTION_BLOCK

// ---- POUs/FB_StepperCtrl.TcPOU
FUNCTION_BLOCK FB_StepperCtrl
VAR
// Axis 1 Stepper Motor Variables
	Axis					: TC2_MC2.AXIS_REF;			(* Reference the one axis being controlled *)
	fbPower_Axis			: MC_Power;					(* FB handles the drive power activation *)
	fbReset_Axis			: MC_Reset;					(* FB Resets the Axis *)
	fbHalt_Axis				: MC_Halt;					(* FB performs an axis halt operation *)
	fbStop_Axis				: MC_Stop;					(* FB performs an axis Stop operation *)
	fbJog_Axis				: MC_Jog;					(* FB allows to jog the axis CW or CCW *)
	fbRead_Position_Axis	: MC_ReadActualPosition;	(* FB reads the axis current position *)
	fbRead_Velocity_Axis	: MC_ReadActualVelocity;	(* FB reads the axis current velocity *)	
	fbSet_Position			: MC_SetPosition;
	fbMove_Absolute_Axis	: MC_MoveAbsolute;			(* FB carries out the axis absolute positioning *)
	fbMove_Relative_Axis	: MC_MoveRelative;

// Misc Variables
	goto_position			: LREAL;
END_VAR
VAR_INPUT
// Power Axis Input Variables
	bEnable					: BOOL;

// Reset Axis Input Variables
	bResetExe				: BOOL;
	
// Halt Axis Input Options
	bHaltExe				: BOOL;
	haltDecel				: LREAL;

// Stop Axis Input Variables
	bStopExe				: BOOL;
	bStopDecel				: LREAL;
	bStopJerk				: LREAL;

// Jog Axis Input Variables
	bJogFwd					: BOOL;
	bJogBack				: BOOL;
	jogPos					: LREAL;
	jogVel					: LREAL := 100;
	jogAccel				: LREAL := 10000;
	jogDecel				: LREAL := 10000;
	jogJerk					: LREAL := 60000;

// Set Position Input Variables
	bSetPosExe				: BOOL;
	setPosPost				: LREAL;

// Move Absolute Input Variables
	bMoveAbsExe				: BOOL;
	moveAbsPosition			: LREAL;
	moveAbsVel				: LREAL;
	moveAbsAccel			: LREAL := 10000;
	moveAbsDecel			: LREAL := 10000;
	moveAbsJerk				: LREAL := 60000;

// Relative Move Input Variables
	bMoveRelExe				: BOOL;
	moveRelDistance			: LREAL;
	moveRelVel				: LREAL;
	moveRelDist				: LREAL;
	moveRelAccel			: LREAL := 10000;
	moveRelDecel			: LREAL := 10000;
	moveRelJerk				: LREAL := 60000;
	
// Misc Input Variables
	sPosition				: STRING;
END_VAR
VAR_OUTPUT
// Power Axis Output Variables
	bPwrStatus				: BOOL;
	
// Reset Axis Output Variables
	bResetDone				: BOOL;
	bResetBusy				: BOOL;
	bResetError				: BOOL;
	resetErrorID			: UDINT;
	
// Halt Axis Output Variables
	bHaltDone				: BOOL;
	bHaltBusy				: BOOL;
	bHaltActive				: BOOL;
	bHaltCmdabort			: BOOL;
	bHaltError				: BOOL;
	haltErrorID				: UDINT;
	
// Stop Axis Output Variables
	bStopDone				: BOOL;
	bStopBusy				: BOOL;
	bStopActive				: BOOL;
	bStopCmdAbort			: BOOL;
	bStopError				: BOOL;
	stopErrorId				: UDINT;
	
// Jog Axis Output Variables
	bJogDone				: BOOL;
	bJogBusy				: BOOL;
	bJogActive				: BOOL;
	bJogAbort				: BOOL;
	bJogError				: BOOL;
	jogErrorID				: UDINT;
	
// Read Position Output Variables
	readPosActPosition		: LREAL;
	
// Read Velocity Output Variables
	readVelActVel			: LREAL;
	
// Set Position Output Variables
	bSetPosDone				: BOOL;
	bSetPosBusy				: BOOL;
	bSetPosError			: BOOL;
	SetPosErrorId			: UDINT;
	
// Move Absolute Output Variables
	bMoveAbsDone			: BOOL;
	bMoveAbsBusy			: BOOL;
	bMoveAbsActive			: BOOL;
	bMoveAbsAbort			: BOOL;
	bMoveAbsError			: BOOL;
	bMoveErrorID			: UDINT;
	
// Move Relative Output Variables
	bMoveRelDone			: BOOL;
	bMoveRelBusy			: BOOL;
	bMoveRelActive			: BOOL;
	bMoveRelCmdAbort		: BOOL;
	bMoveRelError			: BOOL;
	moveRelErrorID			: UDINT;
END_VAR

///////////////////////////////////////////
// AXIS CONTROL
///////////////////////////////////////////

//moveRelDist := STRING_TO_LREAL(sPosition);

(* Enable signals are set *)
fbPower_Axis(
	Axis			:=	Axis,
	Enable			:=	bEnable,
	Enable_Positive	:= 	bEnable,
	Enable_Negative	:= 	bEnable,
	Override		:=	100.000,
	BufferMode		:=	,
	Options			:=	,
	Status			=>	bPwrStatus,
	Busy			=>	,
	Active			=>	,	
	Error			=>	,
	ErrorID			=>	);

(* Axis Reset *)
fbReset_Axis(
	Axis	:= 	Axis,
	Execute	:=	bResetExe,
	Done	=>	bResetDone,
	Busy	=>	bResetBusy,
	Error	=>	bResetError,
	ErrorID	=>	resetErrorID
);
(*
(* Check if Reset was done successfully *)
IF bReset_Done THEN
	bReset := FALSE;
	bMove_Absolute := FALSE;
	bMove_Jog := FALSE;
END_IF	
*)

(* Axis Halt *)
fbHalt_Axis(
	Axis			:= Axis,
	Execute			:= bHaltExe,
	Deceleration	:= haltDecel,
//	Jerk			:= lrJerk_Axis,
	BufferMode		:= MC_Aborting,
	Options			:= ,
	Done			=> bHaltDone,
	Busy			=> bHaltBusy,
	Active			=> bHaltActive,
	CommandAborted	=> bHaltCmdabort,
	Error			=> bHaltError,
	ErrorId			=> haltErrorID	
);
(*	
(* Check if Halt was done successfully *)
IF fbHalt.Done THEN
	bHalt 			:=	FALSE;
	bMove_Absolute	:=	FALSE;
	bMove_Jog		:=	FALSE;
	bTest			:=  TRUE;
END_IF
*)
	
(* Axis Stop *)
fbStop_Axis(
	Axis			:=	Axis,
	Execute			:=	bStopExe,
	Deceleration	:=	bStopDecel,
	Jerk			:=	bStopJerk,
	Options			:=	,
	Done			=>	bStopDone,
	Busy			=>	bStopBusy,
	Active			=>	bStopActive,
	CommandAborted	=>	bStopCmdAbort,
	Error			=>	bStopError,
	ErrorId			=> stopErrorId	
);		

	
(* Axis Jog. bJogFwd true is CW and bJogBack true is CCW *)
fbJog_Axis(
	Axis			:= 	Axis,
	JogForward		:= 	bJogFwd,
	JogBackwards	:= 	bJogBack,
	Mode			:=	MC_JOGMODE_STANDARD_FAST,
	Position		:=	jogPos,
	Velocity		:= 	jogVel,
	Acceleration	:= 	jogAccel,
	Deceleration	:= 	jogDecel,
	Jerk			:= 	jogJerk,
	Done			=>	bJogDone,
	Busy			=>	bJogBusy,
	Active			=>	bJogActive,
	CommandAborted	=> 	bJogAbort,
	Error			=> 	bJogError,
	ErrorId			=> 	jogErrorID
);

(* Get the current Position *)
fbRead_Position_Axis(
	Axis		:= 	Axis,
	Enable		:= 	TRUE,
	Valid		=>	,
	Busy		=> 	,
	Error		=> 	,
	ErrorID		=> 	,
	Position	=>	readPosActPosition
);

(* Get the current Velocity *)
fbRead_Velocity_Axis(
	Axis			:= 	Axis,
	Enable			:= 	TRUE,
	Valid			=>	,
	Busy			=> 	,
	Error			=> 	,
	ErrorID			=> 	,
	ActualVelocity	=>	readVelActVel
);

fbSet_Position(
	Axis := Axis,
	Execute := bSetPosExe,
	Position := setPosPost,
	Mode := FALSE,
	Done => bSetPosDone,
	Busy => bSetPosBusy,
	Error => bSetPosError,
	ErrorId => SetPosErrorID
);

(* Perform an Absolute Motion *)
fbMove_Absolute_Axis(
	Axis			:=	Axis,
	Execute			:= 	bMoveAbsExe,
	Position		:= 	moveAbsPosition,
	Velocity		:= 	moveAbsVel,
	Acceleration 	:= 	moveAbsAccel,
	Deceleration 	:= 	moveAbsDecel,
	Jerk			:= 	moveAbsJerk,
	BufferMode		:=	,
	Options			:=	,
	Done			=>	bMoveAbsDone,
	Busy			=>	bMoveAbsBusy,
	Active			=>	bMoveAbsActive,
	CommandAborted	=>	bMoveAbsAbort,
	Error			=>	bMoveAbsError,
	ErrorID			=>	bMoveErrorID,
);

fbMove_Relative_Axis(
	Axis := Axis,
	Execute := bMoveRelExe,
	Distance := moveRelDist,
	Velocity := moveRelVel,
	Acceleration := moveRelAccel,
	Deceleration := moveRelDecel,
	Jerk := moveRelJerk,
	BufferMode := ,
	Options := ,
	Done => bMoveRelDone,
	Busy => bMoveRelBusy,
	Active => bMoveRelActive,
	CommandAborted => bMoveRelCmdAbort,
	Error => bMoveRelError,
	ErrorID => moveRelErrorID
);

(*
(* Turn off all flags if axis not enabled *)
IF NOT bEnable THEN
	bReset			:=	FALSE;
	bHalt			:=	FALSE;
//	bMove_Absolute	:=	FALSE;
	bMove_Jog		:=	FALSE;
END_IF
*)
(*
(* Turn off all flags if axis not enabled *)
IF (bJogFwd = FALSE AND bJogBack = FALSE) THEN //OR bMove_Absolute = FALSE THEN
//	bStop			:=	TRUE;
	bHalt			:=	TRUE;
//	bMove_Absolute	:=	FALSE;
	bMove_Jog		:=	FALSE;
ELSE
//	bStop			:=	FALSE;
	bHalt			:=	FALSE;
END_IF
*)

END_FUNCTION_BLOCK

// ---- POUs/FB_FanWriteReg.TcPOU
FUNCTION_BLOCK FB_FanWriteReg
VAR_INPUT
	f_mbMaster			: ModbusRtuMaster_KL6x22B;
	f_mbUnit			: BYTE;
	f_mbWriteAddr 		: WORD;
	f_mbWriteData 		: WORD;
END_VAR

VAR_OUTPUT
	f_mbErrorFlag		: BOOL;
	f_mbErrorId			: MODBUS_ERRORS;
	f_mbBusy			: BOOL;
	f_mbBytesRec		: UINT;	
	f_state				: UINT;
	f_nextState			: UINT;
END_VAR

VAR
	
END_VAR

// write register

	f_mbMaster.WriteSingleRegister(
		UnitID := f_mbUnit, 
		Quantity := 1, 
		MBAddr := f_mbWriteAddr, 
		cbLength := SIZEOF(f_mbWriteData), 
		pMemoryAddr := ADR(f_mbWriteData), 
		Execute := TRUE, 
		Timeout := T#1S, 
		BUSY => f_mbBusy, 
		Error => f_mbErrorFlag, 
		ErrorId => f_mbErrorId, 
		cbRead => f_mbBytesRec
	);

	// write complete
	IF f_mbBusy = FALSE THEN
		// reset comms
		f_mbMaster.ReadRegs(Execute := FALSE);
		f_nextState := 1;
		f_state := f_nextState;
		// catch error
		IF f_mbErrorFlag = TRUE THEN
			f_state := 4;
		END_IF
	END_IF

END_FUNCTION_BLOCK

// ---- POUs/FB_ModBusTCPWriteRegs.TcPOU
FUNCTION_BLOCK FB_ModBusTCPWriteRegs
VAR_INPUT
    sIPAddr    			: STRING(15);
    nTCPPort   			: UINT:= MODBUS_TCP_PORT;
    nUnitID    			: BYTE:=16#FF;
    nQuantity  			: WORD;
    nMBAddr    			: WORD;
    cbLength   			: UDINT;
    pDestAddr  			: POINTER TO BYTE;
    bExecute   			: BOOL;
    tTimeout   			: TIME;
END_VAR 
VAR_OUTPUT
    bBUSY      			: BOOL;
    bError     			: BOOL;
    nErrId     			: UDINT;
    cbRead     			: UDINT;
END_VAR 
VAR
    fbWriteRegs        	: FB_MBWriteRegs;
    bReadRegs         	: BOOL;
    bReadRegsBusy     	: BOOL;
    bReadRegsError    	: BOOL;
    nReadRegsErrorId  	: UDINT;
    nReadRegsCount    	: UDINT;
    arrData2           	: ARRAY [1..2] OF WORD;
END_VAR

fbWriteRegs(
	sIPAddr := sIPAddr,						//Is a string containing the IP address of the target device
	nTCPPort := MODBUS_TCP_PORT,			//Port number of the target device
	nUnitID := 255,							//Identification number of a serial sub-network device, 16$FF if TCP/IP is used
	nQuantity := 2,							//Number of output registers (data words) to be write. The value of nQuantity must be > 0
	nMBAddr := 0,							//Start address of the output registers to be write (word offset)
	cbLength := SIZEOF(arrData2),			//Contains the max. byte size of the source buffer. T
	pSrcAddr := ADR(arrData2),				//Contains the address of the source buffer containing the data to be written
	bExecute := fbWriteRegs.bExecute,		//The function block is activated by a rising edge at this input.
	tTimeout := T#1S,						//States the length of the timeout that may not be exceeded by execution of the ADS command
	bBusy => fbWriteRegs.bBusy,				//When the function block is activated this output is set
	bError => fbWriteRegs.bError,			//If an ADS error should occur during the transfer of the command
	nErrId => fbWriteRegs.nErrId				//Supplies the ADS error number when the bError output is set
	);

END_FUNCTION_BLOCK

// ---- GlobalTextList.TcGTLO
TEXTLIST GlobalTextList
  120 = '# STEPS/MOVE TO'
  422 = '#1'
  201 = '#2'
  404 = '%s'
  9 = 'ABSOLUTE MOVE'
  444 = 'ACTUAL POSITION'
  237 = 'ANALOG IN'
  921 = 'ANALOG INPUTS'
  80 = 'AXIS 1'
  339 = 'AXIS 2'
  333 = 'carol E2V05BWB00'
  318 = 'CCMT 4'
  954 = 'CCMT 4 Valve'
  271 = 'Coms Error'
  824 = 'Configuration...'
  90 = 'Current Step Pos.'
  616 = 'E2V05BWB00'
  341 = 'EL7031 CONTROL'
  134 = 'Execute Move'
  915 = 'Execute Movo'
  452 = 'Execute Movove'
  458 = 'EXIT'
  539 = 'Fan Control'
  466 = 'GVL.ai01'
  612 = 'Jog Backwards'
  513 = 'Jog Forwards'
  861 = 'Label'
  472 = 'MAIN.s1'
  846 = 'MOVE TO POSITION'
  753 = 'MOVE TO POSITION:'
  707 = 'Move to Step Pos.'
  142 = 'NEGATIVE  -  POSITIVE'
  457 = 'POSITION'
  253 = 'Pressure [Bar]'
  95 = 'RELATIVE MOVE'
  997 = 'RELAY CTRL'
  177 = 'RTD Temp 1'
  931 = 'RTD Temp 2'
  967 = 'RTD Temp 3'
  233 = 'RTD Temp 4'
  356 = 'RTD Temp 5'
  231 = 'RTD Temperature'
  186 = 'Set RPM'
  971 = 'Setup'
  296 = 'Speed, Nom.'
  181 = 'STEPS TO MOVE'
  541 = 'STEPS TO MOVE/MOVE TO POSITIO+N'
  24 = 'Tachometer'
  525 = 'TC Temperature'
  761 = 'TC Temperature Reading'
  2 = 'Temp 1'
  856 = 'Temp 2'
  146 = 'Temp 3'
  214 = 'Temp 4'
  174 = 'Temp 5'
  25 = 'Temperature'
  668 = 'Temperature [C]'
  254 = 'text'
  236 = 'Thermocouple Temperature Reading'
  881 = 'Valve Control'
  549 = 'Valve Ctrl'
  655 = 'Valve OD (%)'
  89 = 'Vapor Quality'
  827 = 'Vapor Quality Sensor'
END_TEXTLIST

// ---- VISUs/Visu_MAIN.TcVIS
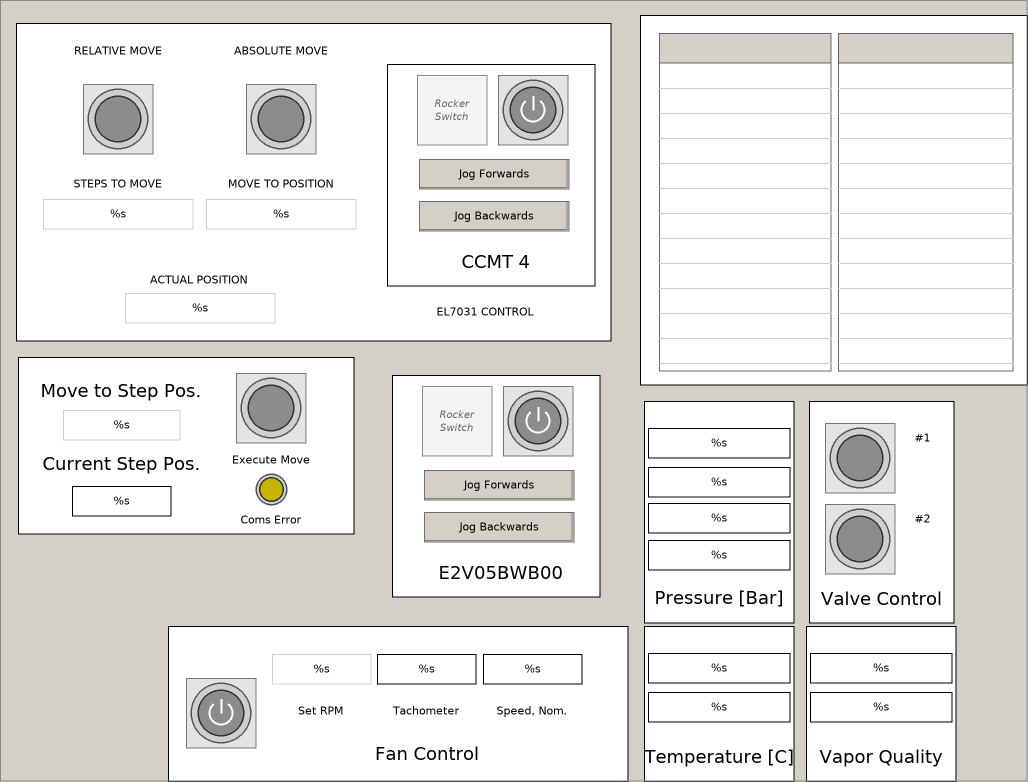
VISUALIZATION Visu_MAIN  // 1028x782
    RoundedRectangle (18,357 336x177)
    Group (392,375 208x222)
        RoundedRectangle (0,0 208x222)
        Button (32,95 150x30), "Jog Forwards"
            tap MAIN.fbAxis2.bJogFwd
        Button (32,137 150x30), "Jog Backwards"
            tap MAIN.fbAxis2.bJogBack
        PowerSwitch (111,11 70x70), variable: MAIN.fbAxis2.bReset, behaviour: TOGGLE, style: Switch-PowerSwitch-Gray
        RockerSwitch (30,11 70x70), variable: MAIN.fbAxis2.bEnable, behaviour: TOGGLE, style: Switch-RockerSwitch-Gray
        Label (34,180 150x36), "E2V05BWB00"
    Group (809,401 145x222)
        RoundedRectangle (0,0 145x222)
        PushSwitchLed (16,22 70x70), variable: bRelay1, behaviour: TOGGLE, style: Switch-PushSwitchLed-Gray
        PushSwitchLed (16,103 70x70), variable: bRelay2, behaviour: TOGGLE, style: Switch-PushSwitchLed-Gray
        Label (7,180 131x36), "Valve Control"
        Label (89,22 49x30), "#1"
        Label (89,103 49x30), "#2"
    Group (644,401 150x222)
        RoundedRectangle (0,0 150x222)
        Label (7,179 136x36), "Pressure [Bar]"
        Rectangle (4,27 142x30), "%s", text variable: MAIN.sPress01
        Rectangle (4,66 142x30), "%s", text variable: MAIN.sPress02
        Rectangle (4,102 142x30), "%s", text variable: MAIN.sPress03
        Rectangle (4,139 142x30), "%s", text variable: MAIN.sPress04
    Group (644,626 150x156)
        RoundedRectangle (0,0 150x156)
        Label (4,113 143x36), "Temperature [C]"
        Rectangle (4,27 142x30), "%s", text variable: MAIN.SurfaceRTD1
        Rectangle (4,66 142x30), "%s", text variable: MAIN.SurfaceRTD2
    Group (806,626 150x156)
        RoundedRectangle (0,0 150x156)
        Label (7,113 136x36), "Vapor Quality"
        Rectangle (4,27 142x30), "%s", text variable: MAIN.sVaporQual
        Rectangle (4,66 142x30), "%s", text variable: MAIN.sPress02
    RoundedRectangle (640,15 388x370)
    Table (659,33 172x338), data array: MAIN.fbFormatRTD.RTDarray
        p3854506369: MAIN.fbFormatRTD.RTDarray[INDEX]
        p2232123230: RTD Temperature
    Table (838,33 175x338), data array: MAIN.fbmVtoTemp.degCtempArray
        p3854506369: MAIN.fbmVtoTemp.degCtempArray[INDEX]
    RoundedRectangle (168,626 460x156)
    Label (359,736 136x36), "Fan Control"
    PowerSwitch (186,678 70x70), variable: MAIN.bFanEnable, behaviour: TOGGLE, style: Switch-PowerSwitch-Gray
    Label (273,693 96x36), "Set RPM"
    Rectangle (377,654 99x30), "%s", text variable: MAIN.Fan1.f_tachometerData
    Label (378,693 96x36), "Tachometer"
    Rectangle (483,654 99x30), "%s", text variable: MAIN.Fan1.f_speedNominal
    Label (484,693 96x36), "Speed, Nom."
    Textfield (272,654 99x30), "%s", text variable: MAIN.smbRPM
        OnMouseDown: write the text variable via Default
    Group (16,23 595x318)
        RoundedRectangle (0,0 595x318)
        Textfield (109,270 150x30), "%s", text variable: MAIN.fbAxis1.fbRead_Position_Axis.Position
            OnMouseDown: write the text variable via Default
        Label (108,242 150x30), "ACTUAL POSITION"
        PushSwitch (67,61 70x70), variable: MAIN.bMoveRelative, behaviour: TOGGLE, style: Switch-PushSwitch-Gray
        Label (27,13 150x30), "RELATIVE MOVE"
        Textfield (27,176 150x30), "%s", text variable: MAIN.sStepperNumSteps
            OnMouseClick: write the text variable via Default
        Label (27,146 150x30), "STEPS TO MOVE"
        Group (190,13 150x118)
            PushSwitch (40,48 70x70), variable: MAIN.bMoveAbsolute, behaviour: TOGGLE, style: Switch-PushSwitch-Gray
            Label (0,0 150x30), "ABSOLUTE MOVE"
        Label (190,146 150x30), "MOVE TO POSITION"
        Textfield (190,176 150x30), "%s", text variable: MAIN.sStepperGoTo
            OnMouseClick: write the text variable via Default
        RoundedRectangle (371,41 208x222)
        Button (403,136 150x30), "Jog Forwards"
            tap MAIN.bJogFwd
        Button (403,178 150x30), "Jog Backwards"
            tap MAIN.bJogBack
        PowerSwitch (482,52 70x70), variable: MAIN.fbAxis1.bResetExe, behaviour: TOGGLE, style: Switch-PowerSwitch-Gray
        RockerSwitch (401,52 70x70), variable: MAIN.fbAxis1.bEnable, behaviour: TOGGLE, style: Switch-RockerSwitch-Gray
        Label (405,221 150x36), "CCMT 4"
    PushSwitch (236,373 70x70), variable: MAIN.btnMbActivate, behaviour: TOGGLE, style: Switch-PushSwitch-Gray
    Label (410,297 150x30), "EL7031 CONTROL"
    Textfield (63,410 117x30), "%s", text variable: MAIN.percentOD
        OnMouseDown: write the text variable via Default
    Rectangle (72,486 99x30), "%s", text variable: MAIN.sCCMTPos
    Label (31,373 180x36), "Move to Step Pos."
    Label (42,446 159x36), "Current Step Pos."
    Lamp1 (251,471 41x37), variable: MAIN.fbCCMT4mb.f_mbErrorFlag, style: Lamp-Lamp1-Yellow
    Label (223,502 96x36), "Coms Error"
    Label (223,442 96x36), "Execute Move"
END_VISUALIZATION
